// TwinCAT 3 PLC project Belsignaal_FD
// ProgramVersion: 3.1.4024.0
// libraries:
//   Tc2_Standard, * (Beckhoff Automation GmbH)
//   Tc2_System, * (Beckhoff Automation GmbH)
//   Tc3_Module, * (Beckhoff Automation GmbH)
// project tree:
//   / PlcTask.TcTTO
//   POUs/ MAIN.TcPOU
// (motion and I/O tree: see PLC project trappenhuis_extraverlenging)
// real-time tasks:
//   TASK PlcTask: cycle T#10ms, priority 20, ADS port 350
//   TASK PlcTask1: cycle T#10ms, priority 21, ADS port 351
//   TASK PlcTask2: cycle T#10ms, priority 22, ADS port 352
//   TASK PlcTask3: cycle T#10ms, priority 23, ADS port 353
//   TASK PlcTask4: cycle T#10ms, priority 24, ADS port 354
//   TASK PlcTask5: cycle T#10ms, priority 25, ADS port 355
//   TASK PlcTask6: cycle T#10ms, priority 26, ADS port 356
//   TASK PlcTask7: cycle T#10ms, priority 27, ADS port 357
//   TASK PlcTask8: cycle T#10ms, priority 28, ADS port 358
//   TASK PlcTask9: cycle T#10ms, priority 29, ADS port 359
//   TASK PlcTask10: cycle T#10ms, priority 30, ADS port 360

CONFIGURATION Belsignaal_FD
    RESOURCE PLC ON TwinCAT3
        TASK PlcTask(INTERVAL := T#10ms, PRIORITY := 28);
        PROGRAM MAIN WITH PlcTask : MAIN;
    END_RESOURCE
END_CONFIGURATION

// ---- POUs/MAIN.TcPOU
PROGRAM MAIN
VAR
	// Digitale ingangen
	bSensor1 AT %I*: BOOL;
	bSensor2 AT %I*: BOOL;
	bReset   AT %I*: BOOL;
	
	// Digitale uitgangen
	bZoemer  AT %Q*: BOOL;
	
	// Functies
	NaarBinnen: R_TRIG;
	Aantalklanten: CTU;
	ZoemerLimit: TOF;
END_VAR

(*
Belsignaal aan winkeldeur (3 regel code +1 + 1)

elke uitbreiding voegt 1 regel code toe op de basis 3 regels code voor de eerste opdracht 

    Aan de ingangsdeur van een winkel staan twee fotocellen S01 en S02 opgesteld.
    Wanneer een klant binnenkomt wordt eerst S01 onderbroken, daarna S02, een bel of zoemer zal in werking treden zolang de lichtstralen van de fotocellen onderbroken zijn.
    Wanneer een klant buitengaat wordt eerst S02 onderbroken, daarna S01, hier mag de bel of zoemer niet werken.

Uitbreiding: Tel het aantal binnenkomende klanten met een counter FB.

Uitbreiding: Om te vermijden dat de bel blijft rinkelen als een klant aan de deur blijft stilstaan zal de bel of zoemer slechts 0,5 seconde werken
*)

// niet zeker 2e uitbreiding

NaarBinnen(CLK:=bSensor2 , Q=> );
bZoemer S=(bSensor1 AND NaarBinnen.Q);
bZoemer R=((NOT bSensor1) AND (NOT bSensor2)OR(ZoemerLimit.Q));

// Uitbreiding 1
Aantalklanten(CU:=(bSensor1 AND NaarBinnen.Q), RESET:=bReset);

// Uitbreiding 2
ZoemerLimit(IN:=(bSensor1 AND NaarBinnen.Q), PT:=T#5S , Q=>bZoemer , ET=> );

END_PROGRAM
